FUNCTION_BLOCK FB_HomeWriteNcVelocities
VAR_INPUT
    En: BOOL;
    bReset: BOOL;
    bExecute: BOOL;
    fVelocityToCam: LREAL;
    fVelocityFromCam: LREAL;
END_VAR
VAR_IN_OUT
    Axis: AXIS_REF;
END_VAR
VAR_OUTPUT
    EnO: BOOL;
    bBusy: BOOL;
    bDone: BOOL;
    bError: BOOL;
    nErrorId: UDINT;
END_VAR
VAR
    fbExecuteRiseEdge: R_TRIG;
    fbWriteVelocityToCam:FB_WriteFloatParameter;
    fbWriteVelocityFromCam:FB_WriteFloatParameter;
END_VAR

En:=EnO;
IF bReset THEN
    bError:=FALSE;
    nErrorId:=0;
END_IF

fbExecuteRiseEdge(CLK:=bExecute);

fbWriteVelocityToCam(
    bExecute:=bExecute,
    nDeviceGroup:= 16#4000,
    nIndexOffset:= 16#6,
    nData:=fVelocityToCam,
    Axis:= Axis);

fbWriteVelocityFromCam(
    bExecute:=bExecute,
    nDeviceGroup:= 16#4000,
    nIndexOffset:= 16#7,
    nData:=fVelocityFromCam,
    Axis:= Axis);

bBusy:=fbWriteVelocityFromCam.bBusy OR fbWriteVelocityToCam.bBusy;
bDone:=fbWriteVelocityFromCam.bDone AND fbWriteVelocityToCam.bDone AND bExecute;

bError:=fbWriteVelocityToCam.bError OR fbWriteVelocityFromCam.bError;
IF fbWriteVelocityToCam.bError THEN
  nErrorId:=fbWriteVelocityToCam.nErrorId;
ELSIF fbWriteVelocityFromCam.bError THEN
  nErrorId:=fbWriteVelocityFromCam.nErrorId;
END_IF

END_FUNCTION_BLOCK

(* stored: Version 1.1.0.1, ProductVersion 3.1.4024.0
   POU FB_HomeWriteNcVelocities: Id {db235f88-cc6a-42fd-a27f-0c03a858adf6}, SpecialFunc None *)
